// SIMATIC S7-200 project (STEP 7-Micro/WIN), CPU 224XP REL 02.01

SYMBOL_TABLE USER1
light_switch     I0.0     // turn on/off light
stop_EMG         I0.5     // EMG stop
sleep_state      M0.1     // sleep status
D1               Q0.0     // light
END_SYMBOL_TABLE

ORGANIZATION_BLOCK MAIN:OB1
TITLE=PROGRAM COMMENTS
BEGIN
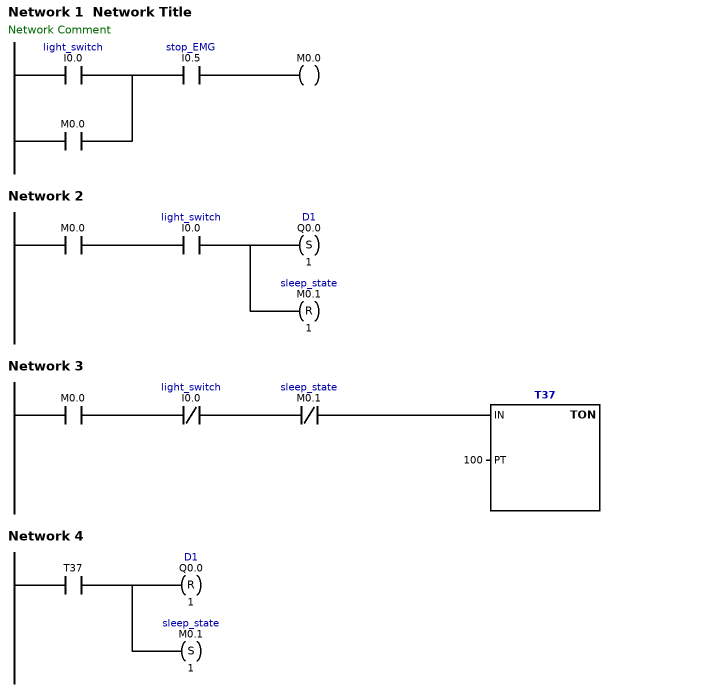
Network 1 // Network Title
// Network Comment
LD     light_switch:I0.0
O      M0.0
A      stop_EMG:I0.5
=      M0.0
Network 2
LD     M0.0
A      light_switch:I0.0
S      D1:Q0.0, 1
R      sleep_state:M0.1, 1
Network 3
LD     M0.0
AN     light_switch:I0.0
AN     sleep_state:M0.1
TON    T37, 100
Network 4
LD     T37
R      D1:Q0.0, 1
S      sleep_state:M0.1, 1
END_ORGANIZATION_BLOCK
